// TIA Portal project "teknofest" (V14)

(* hardware
DEVICE "S7-1200 station_1"  S7-1200 Station
   slot 0: "Rack_0"  S7-1200 Rack  Rack  V1.0
   slot 1: "PLC_1"  CPU 1214C DC/DC/DC  6ES7 214-1AG40-0XB0  V4.2
DEVICE "HMI_1"  KTP700 Basic PN
   slot 0: "KTP700 Basic PN"  KTP700 Basic PN  6AV2 123-2GB03-0AX0  14.0.0.0
   slot 1: "HMI_RT_1"  KTP700 Basic PN  6AV2 123-2GB03-0AX0  14.0.0.0
   slot 5: "HMI_1.IE_CP_1"  PROFINET Interface  14.0.0.0
      slot 1: "PROFINET Interface_1"  PROFINET Interface
         slot 1: "Port_1"  Port
*)

// ===== PLC "PLC_1"  CPU 1214C DC/DC/DC =====

VAR_GLOBAL   // PLC tag table "Default tag table"
   "ACİL STOP" AT %I0.0 : Bool;
   "STOP_S2" AT %I0.2 : Bool;
   "START_S1" AT %I0.1 : Bool;
   "MOTOR_K1" AT %Q0.0 : Bool;
   "SİSTEM AKTİF" AT %M0.0 : Bool;
   "HMI_START" AT %M0.1 : Bool;
   "SENSÖR_BP1" AT %I1.0 : Bool;
   "YEŞİL_SİNYAL_K5" AT %Q0.4 : Bool;
   "KIRMIZI_SİNYAL_K6" AT %Q0.5 : Bool;
   "ROBOTKOL_BAŞLA_K10" AT %Q1.1 : Bool;
   "SENSÖR_BP2" AT %I1.1 : Bool;
   "SENSÖR_BP3" AT %I1.2 : Bool;
   "SENSÖR_BP4" AT %I1.3 : Bool;
   "HMI_STOP" AT %M0.2 : Bool;
END_VAR

ORGANIZATION_BLOCK "Main"   // OB1, LAD, ProgramCycle
TITLE = "Main Program Sweep (Cycle)"
{ S7_Optimized_Access := 'TRUE' }
VERSION : 0.1
   VAR_INPUT
      Initial_Call : Bool;   // Initial call of this OB
      Remanence : Bool;   // =True, if remanent data are available
   END_VAR
BEGIN

REGION Network 1: SİSTEM KONTROLÜ
   // SİSTEM DE KONVEYÖR GİRİŞİNDE KÜP ALGILANDIĞINDA OPERATÖR PANELİ VEYA PANO ÜZERİNDEN FİZİKSEL BUTON İLE SİSTEMİN BAŞLATILMASI VE DURDURULMASI.
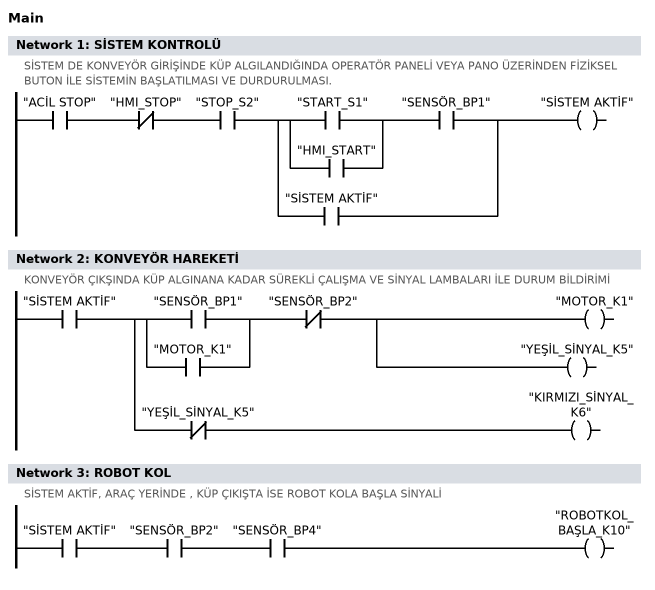
   RUNG wire#powerrail
      Contact( "ACİL STOP" )
      I_Contact( "HMI_STOP" )
      Contact( "STOP_S2" )
      wire#w1
      Contact( "START_S1" )
      wire#w2
      Contact( "SENSÖR_BP1" )
      wire#w3
      Coil( "SİSTEM AKTİF" )
   END_RUNG
   RUNG wire#w1
      Contact( "HMI_START" )
   END_RUNG wire#w2
   RUNG wire#w1
      Contact( "SİSTEM AKTİF" )
   END_RUNG wire#w3
   // the same network as SCL:
   "SİSTEM AKTİF" := "ACİL STOP" AND NOT "HMI_STOP" AND "STOP_S2" AND ((("START_S1" OR "HMI_START") AND "SENSÖR_BP1") OR "SİSTEM AKTİF");
END_REGION

REGION Network 2: KONVEYÖR HAREKETİ
   // KONVEYÖR ÇIKŞINDA KÜP ALGINANA KADAR SÜREKLİ ÇALIŞMA VE SİNYAL LAMBALARI İLE DURUM BİLDİRİMİ
   RUNG wire#powerrail
      Contact( "SİSTEM AKTİF" )
      wire#w1
      Contact( "SENSÖR_BP1" )
      wire#w2
      I_Contact( "SENSÖR_BP2" )
      wire#w3
      Coil( "MOTOR_K1" )
   END_RUNG
   RUNG wire#w1
      Contact( "MOTOR_K1" )
   END_RUNG wire#w2
   RUNG wire#w3
      Coil( "YEŞİL_SİNYAL_K5" )
   END_RUNG
   RUNG wire#w1
      I_Contact( "YEŞİL_SİNYAL_K5" )
      Coil( "KIRMIZI_SİNYAL_K6" )
   END_RUNG
   // the same network as SCL:
   "MOTOR_K1" := "SİSTEM AKTİF" AND ("SENSÖR_BP1" OR "MOTOR_K1") AND NOT "SENSÖR_BP2";
   "YEŞİL_SİNYAL_K5" := "MOTOR_K1";
   "KIRMIZI_SİNYAL_K6" := "SİSTEM AKTİF" AND NOT "YEŞİL_SİNYAL_K5";
END_REGION

REGION Network 3: ROBOT KOL
   // SİSTEM AKTİF, ARAÇ YERİNDE , KÜP ÇIKIŞTA İSE ROBOT KOLA BAŞLA SİNYALİ
   RUNG wire#powerrail
      Contact( "SİSTEM AKTİF" )
      Contact( "SENSÖR_BP2" )
      Contact( "SENSÖR_BP4" )
      Coil( "ROBOTKOL_BAŞLA_K10" )
   END_RUNG
   // the same network as SCL:
   "ROBOTKOL_BAŞLA_K10" := "SİSTEM AKTİF" AND "SENSÖR_BP2" AND "SENSÖR_BP4";
END_REGION
END_ORGANIZATION_BLOCK

(* ===== HMI "HMI_RT_1" =====
system functions are stored by id; their names below are inferred from use
connection "HMI_Connection_1": ETHERNET, SMART_S7_1200_OMS

HMI tags "Default tag table"
   "Tag_ScreenNumber" : UInt, internal
   "MOTOR_K1" : Bool = PLC MOTOR_K1 AT %Q0.0, 1 s
   "ROBOTKOL_BAŞLA_K10" : Bool = PLC ROBOTKOL_BAŞLA_K10 AT %Q1.1, 1 s
   "HMI_START" : Bool = PLC HMI_START AT %M0.1, 100 ms
   "HMI_STOP" : Bool = PLC HMI_STOP AT %M0.2, 100 ms
   "SENSÖR_BP1" : Bool = PLC SENSÖR_BP1 AT %I1.0, 100 ms
   "SENSÖR_BP3" : Bool = PLC SENSÖR_BP3 AT %I1.2, 100 ms
   "SENSÖR_BP2" : Bool = PLC SENSÖR_BP2 AT %I1.1, 100 ms

Template "Template_1" 800x480
   Button "Exit" at 714,429 size 71x50; TextOff 'Exit'; PictureOff "ExitRuntime_KTP700_Basic_PN_TR"; PictureOn "ExitRuntime_KTP700_Basic_PN_TR"
      on Release: StopRuntime(0)
   Button "Log on" at 614,429 size 71x50; TextOff 'Log on'; PictureOff "Login_KTP700_Basic_PN_TR"; PictureOn "Login_KTP700_Basic_PN_TR"
      on Release: function_a2a04561()
   Button "Language" at 514,429 size 71x50; TextOff 'Language'; PictureOff "ToggleLanguage_KTP700_Basic_PN_TR"; PictureOn "ToggleLanguage_KTP700_Basic_PN_TR"
      on Release: function_fb9197e8(-1)
   Button "Template_Button" at 414,429 size 71x50; TextOff 'Text'
   Button "Template_Button_1" at 314,429 size 71x50; TextOff 'Text'
   Button "Template_Button_2" at 214,429 size 71x50; TextOff 'Text'
   Button "Alarms" at 114,429 size 71x50; TextOff 'Alarms'; PictureOff "AlarmDisplay_KTP700_Basic_PN_TR"; PictureOn "AlarmDisplay_KTP700_Basic_PN_TR"
      on Release: function_ef3f5d25("Alarm window_Unacknowledged", -1)
   Button "Start screen" at 14,429 size 71x50; TextOff 'Start screen'; PictureOff "NavigateHome_KTP700_Basic_PN_TR"; PictureOn "NavigateHome_KTP700_Basic_PN_TR"
      on Release: ActivateScreen("ANA EKRAN", 0)
   SymbolicIOField "Symbolic_IO_Field_Screen" at 93,9 size 600x33; TextOff '0'; TextOn '1'; TextList "TextList_ScreenNames"
      ProcessValue <- "Tag_ScreenNumber"
      on Change: ActivateScreenByNumber("Tag_ScreenNumber", 0)
   DateTimeField "HmiScreenItemData" at 695,25 size 105x25
   DateTimeField "HmiScreenItemData_1" at 695,0 size 105x25
   GraphicView "Logo" at 0,0 size 91x51; Picture "Logo of HMI_1"

screen "ANA EKRAN" 800x480, template "Template_1"
   on GenerateScreen: SetTag("Tag_ScreenNumber", 1)
   Button "Button_1" at 35,100 size 150x100; TextOff 'START'
      on Press: SetBit("HMI_START")
      on Release: ResetBit("HMI_START")
   Button "Button_2" at 35,210 size 150x100; TextOff 'STOP'
      on Press: SetBit("HMI_STOP")
      on Release: ResetBit("HMI_STOP")
   Circle "Circle_1" at 311,147 size 46x46
      Appearance <- "MOTOR_K1"
   Circle "Circle_2" at 522,147 size 46x46
      Appearance <- "ROBOTKOL_BAŞLA_K10"
   TextField "Text field_1" at 275,115 size 122x23; Text 'SİSTEM AKTİF'
   TextField "Text field_2" at 463,115 size 159x23; Text 'ROBOT KOL BAŞLA'
   GraphicView "Graphic view_1" at 200,300 size 600x100; Picture "Graphic_2"
   GraphicView "Graphic view_2" at 275,275 size 75x75; Picture "Graphic_3"
      Visibility <- "SENSÖR_BP1"
   GraphicView "Graphic view_3" at 455,275 size 75x75; Picture "Graphic_3"
      Visibility <- "SENSÖR_BP3"
   GraphicView "Graphic view_4" at 635,275 size 75x75; Picture "Graphic_3"
      Visibility <- "SENSÖR_BP2"
*)